// TIA Portal V21 program export: 2 tag tables, 0 data types, 0 data blocks, 2 code blocks (in call order from the OBs), 0 instance data blocks

VAR_GLOBAL   // PLC tag table "Default tag table"
END_VAR

VAR_GLOBAL   // PLC tag table "InputOutput"
   Input_0 AT %I0.0 : Bool;
   Input_1 AT %I0.1 : Bool;
   Input_2 AT %I0.2 : Bool;
   Input_3 AT %I0.3 : Bool;
   Input_4 AT %I0.4 : Bool;
   Input_5 AT %I0.5 : Bool;
   Input_6 AT %I0.6 : Bool;
   Input_7 AT %I0.7 : Bool;
   Input_8 AT %I1.0 : Bool;
   Input_9 AT %I1.1 : Bool;
   Input_10 AT %I1.2 : Bool;
   Input_11 AT %I1.3 : Bool;
   Input_12 AT %I1.4 : Bool;
   Input_13 AT %I1.5 : Bool;
   Output_0 AT %Q0.0 : Bool;
   Output_1 AT %Q0.1 : Bool;
   Output_2 AT %Q0.2 : Bool;
   Output_3 AT %Q0.3 : Bool;
   Output_4 AT %Q0.4 : Bool;
   Output_5 AT %Q0.5 : Bool;
   Output_6 AT %Q0.6 : Bool;
   Output_7 AT %Q0.7 : Bool;
   Output_8 AT %Q1.0 : Bool;
   Output_9 AT %Q1.1 : Bool;
END_VAR

ORGANIZATION_BLOCK "Main"   // OB1, LAD, ProgramCycle
TITLE = "Main Program Sweep (Cycle)"
{ S7_Optimized_Access := 'TRUE' }
// stored: SetENOAutomatically false
   VAR_INPUT
      Initial_Call : Bool;   // Initial call of this OB
      Remanence : Bool;   // =True, if remanent data are available
   END_VAR
BEGIN

REGION Network 1
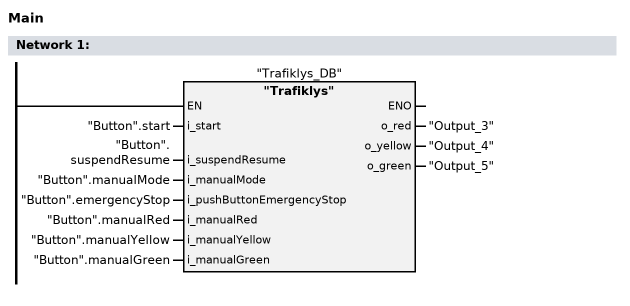
   RUNG wire#powerrail
      "Trafiklys_DB"(i_start := "Button".start, i_suspendResume := "Button".suspendResume, i_manualMode := "Button".manualMode, i_pushButtonEmergencyStop := "Button".emergencyStop, i_manualRed := "Button".manualRed, i_manualYellow := "Button".manualYellow, i_manualGreen := "Button".manualGreen, o_red => "Output_3", o_yellow => "Output_4", o_green => "Output_5")
   END_RUNG
   // the same network as SCL:
   "Trafiklys_DB"(i_start := "Button".start,   // "Trafiklys"
                  i_suspendResume := "Button".suspendResume,
                  i_manualMode := "Button".manualMode,
                  i_pushButtonEmergencyStop := "Button".emergencyStop,
                  i_manualRed := "Button".manualRed,
                  i_manualYellow := "Button".manualYellow,
                  i_manualGreen := "Button".manualGreen,
                  o_red => "Output_3",
                  o_yellow => "Output_4",
                  o_green => "Output_5");
END_REGION

REGION Network 3 (SCL)
   "Button".start := "Input_0";
   "Button".suspendResume := "Input_1";
   "Button".manualMode := "Input_2";
   "Button".emergencyStop := "Input_3";
   "Button".manualRed := "Input_4";
   "Button".manualYellow := "Input_5";
   "Button".manualGreen := "Input_6";
END_REGION
END_ORGANIZATION_BLOCK

FUNCTION_BLOCK "Block_1"
{ S7_Optimized_Access := 'TRUE' }
VERSION : 0.1

BEGIN
	//jeg kan her lave en kommentar som jeg faktisk kan læse
	//
	
END_FUNCTION_BLOCK
